Staubli VAL3: remMovSph.pgx

public program remMovSph(num& nAzi[], num& nEle[], num& nRad[], string& sReturn[])
  local trsf trXYZ
begin
  // Move to designated point in spherical coordinates
  // Point detector to the center of rotation
  //
  logMsg("call remMovSph")
  // Transpose trsf to get correct x, y, z and rotational values
  //trXYZ={0,0,0,0,0,0}
  //trXYZ=trXYZ*{0,0,0,0,nAzi,0}
  //trXYZ=trXYZ*{0,0,0,-nEle,0,0}
  //trXYZ=trXYZ*{0,0,nRad,0,0,0}
  //trXYZ=trXYZ*{0,0,0,-180,0,0}

      // new definitions to match SLAC spec math
    trXYZ={0,0,0,0,0,0}
    // Add AZ component:  rotate about fIPn_+Yaxis
   trXYZ=trXYZ*{0,0,0,0,nAzi,0}
    // Add EL component:  rotate about fIPn_+Z'axis
   trXYZ=trXYZ*{0,0,0,-nEle,0,0}
    // Add RA component:  translate along fIPn+X'axis
    trXYZ=trXYZ*{0,0,nRad,0,0,0}
    // now transform the point so that +Zaxis points back to fIPn
   trXYZ=trXYZ*{0,0,0,0,-180,0}
   //trXYZ.config={sfree,efree,wfree}


  call remMovPoint(trXYZ,sReturn)
end
